{attribute 'GeneratedUsingTerminal: EL1262-0000-0002'}
{attribute addProperty BoxType "EL1262-0000-0002"}
{attribute addProperty Id "Ch2_InputAT %I*BOOL1"}
{attribute addProperty CRC "2024646924"}
{attribute addProperty Size "1"}
TYPE Ch2_Input_78ADA90C :
STRUCT
	{attribute addProperty Name "Ch2_Input"}
	Ch2_Input AT %I* : BOOL;
END_STRUCT
END_TYPE

(* stored: Version 1.2.0.0, ProductVersion 3.1.4024.9
   DUT Ch2_Input_78ADA90C: Id {c0733592-c15c-421e-81b6-831077bb8ac9} *)
